TYPE st_BMS_Set :
STRUCT
	b_enable	: BOOL := TRUE;
	r_SocMax	: REAL := 90;
	r_SocMin	: REAL := 10;
END_STRUCT
END_TYPE

(* stored: Version 1.1.0.1, ProductVersion 3.1.4024.12
   DUT st_BMS_Set: Id {4cb700d9-e364-4d65-b7d9-f966915c7593} *)
